// TIA Portal V20 export
TYPE "typeEt200SpMotorstarterInterfaceHmi"
// stored: Access Published
   STRUCT
      et200SpMotorstarterReadValue : Bool;   // read Value of MotorStarter
      et200SpNumberOfMotorstarters { ExternalWritable := 'False'} : USInt;   // Number of Motor Starters
      et200SpUnitMotorstarter : USInt := 1;   // Unit selected
      et200SpEMMotorstarter : USInt := 0;   // Equipment Module selected
      et200SpMotorstarterCurrent : Array[0.."NO_OF_ET200SPMOTORSTARTER"] of Real;   // Aktuelle Werte / Current values
      et200SpMotorstarterInputs : Array[0.."NO_OF_ET200SPMOTORSTARTER"] of "LSicar_typeMotorstarterIn";   // Motorstarter Data Inputs HMI
      et200SpMotorstarterOutputs : Array[0.."NO_OF_ET200SPMOTORSTARTER"] of "LSicar_typeMotorstarterOut";   // Motorstarter Data Outputs HMI
   END_STRUCT;
END_TYPE
